DATA_BLOCK "DB_BSO40_Template"
TITLE =%version: 0.02 % CN: 20
//History:
//This version  %created_by: nlhdl %
//              %date_created: Friday, March 24, 2017 12:58:03 %
//              %release: VI_RAW/RA_Dev %
//
//Modification History:                                   By:    Date:     Rev:
//----------------------------------------------------  -------  --------  -----
//ra#19216: update DB_BSO40_Template file               nlHdL    24-03-17   0.02
//
FAMILY : General
VERSION : 0.0


  STRUCT
   Coordination_Area : WORD ;	//Coordination area
   Communication_Alive_Sign : INT ;	//Lifesign response
   New_LPN_Present : BOOL ;	//New LPN is present
   Cancel_Encoding : BOOL ;	//Cancel coding button pressed
   Encode_Request : BOOL ;	//Item present which should be encoded
   State_Processing : BOOL ;	//Barcode is being checked for validity
   State_Barcode_Valid : BOOL ;	//Entered barcode is valid
   State_Barcode_Invalid : BOOL ;	//Entered barcode is invalid
   LPN : ARRAY  [0 .. 9 ] OF //Most recent LPN code
   CHAR ;
  END_STRUCT ;
BEGIN
   Coordination_Area := W#16#0;
   Communication_Alive_Sign := 0;
   New_LPN_Present := FALSE;
   Cancel_Encoding := FALSE;
   Encode_Request := FALSE;
   State_Processing := FALSE;
   State_Barcode_Valid := FALSE;
   State_Barcode_Invalid := FALSE;
   LPN[0] := ' ';
   LPN[1] := ' ';
   LPN[2] := ' ';
   LPN[3] := ' ';
   LPN[4] := ' ';
   LPN[5] := ' ';
   LPN[6] := ' ';
   LPN[7] := ' ';
   LPN[8] := ' ';
   LPN[9] := ' ';
END_DATA_BLOCK

